// TIA Portal project "TesisIsitma_v1" (V19)

(* hardware
DEVICE "S7-1200 station_1"  S7-1200 Station
   slot 0: "Rack_0"  S7-1200 Rack  Rack  V1.0
   slot 1: "PLC_1"  CPU 1215C DC/DC/DC  6ES7 215-1AG40-0XB0  V4.5
*)

// ===== PLC "PLC_1"  CPU 1215C DC/DC/DC =====

VAR_GLOBAL   // PLC tag table "Default tag table"
   "System_Byte" AT %MB1 : Byte;
   "FirstScan" AT %M1.0 : Bool;
   "DiagStatusUpdate" AT %M1.1 : Bool;
   "AlwaysTRUE" AT %M1.2 : Bool;
   "AlwaysFALSE" AT %M1.3 : Bool;
   "Clock_Byte" AT %MB0 : Byte;
   "Clock_10Hz" AT %M0.0 : Bool;
   "Clock_5Hz" AT %M0.1 : Bool;
   "Clock_2.5Hz" AT %M0.2 : Bool;
   "Clock_2Hz" AT %M0.3 : Bool;
   "Clock_1.25Hz" AT %M0.4 : Bool;
   "Clock_1Hz" AT %M0.5 : Bool;
   "Clock_0.625Hz" AT %M0.6 : Bool;
   "Clock_0.5Hz" AT %M0.7 : Bool;
   "xSim" AT %M2.0 : Bool;
END_VAR

DATA_BLOCK "DB_Modbus"   // DB2
{ S7_Optimized_Access := 'FALSE' }
VERSION : 0.1
   VAR
      Req : Bool;
      Disconnect : Bool;
      Mode : USInt;
      DataAddress : UDInt := 40001;
      DataLength : UInt := 2;
      DataPointer : Array[0..3] of Byte;
      Connect : TCON_IP_v4;
   END_VAR
BEGIN
   Connect.RemoteAddress.ADDR[1] := 192;
   Connect.RemoteAddress.ADDR[2] := 168;
   Connect.RemoteAddress.ADDR[3] := 0;
   Connect.RemoteAddress.ADDR[4] := 48;
   Connect.InterfaceId := 64;
   Connect.ID := 6;
   Connect.RemotePort := 502;
   Connect.LocalPort := 502;
   Connect.ActiveEstablished := 1;
END_DATA_BLOCK

DATA_BLOCK "DB_Trig"   // DB3
{ S7_Optimized_Access := 'TRUE' }
VERSION : 0.1
   VAR
      "1" : Bool;
      "2" : Bool;
      "3" : Bool;
      "4" : Bool;
      "5" : Bool;
      "6" : Bool;
      "7" : Bool;
      "8" : Bool;
      "9" : Bool;
      "10" : Bool;
   END_VAR
BEGIN
END_DATA_BLOCK

ORGANIZATION_BLOCK "Main"   // OB1, LAD, ProgramCycle
TITLE = "Main Program Sweep (Cycle)"
{ S7_Optimized_Access := 'TRUE' }
VERSION : 0.1
   VAR_INPUT
      Initial_Call : Bool;   // Initial call of this OB
      Remanence : Bool;   // =True, if remanent data are available
   END_VAR
   VAR_TEMP   // added for the SCL form of the ladder/FBD networks
      _w1 : Bool;
      _w2 : Bool;
   END_VAR
BEGIN

REGION Network 1
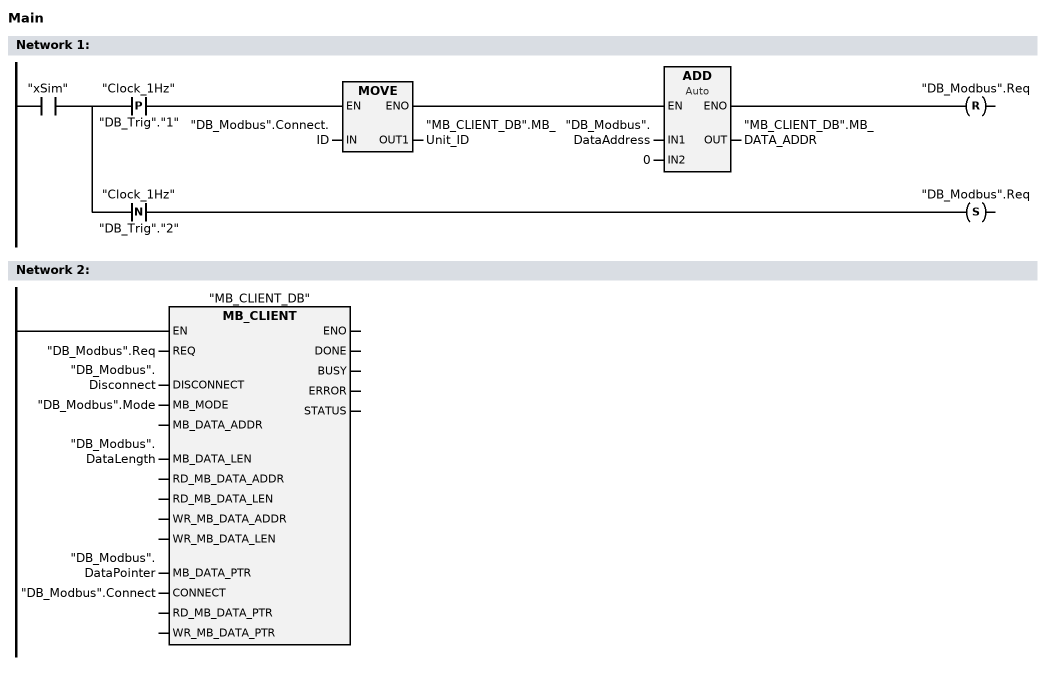
   RUNG wire#powerrail
      Contact( "xSim" )
      wire#w1
      P_Contact(operand := "Clock_1Hz", bit := "DB_Trig"."1")
      Move(in := "DB_Modbus".Connect.ID, out1 => "MB_CLIENT_DB".MB_Unit_ID)
      Add(in1 := "DB_Modbus".DataAddress, in2 := 0, out => "MB_CLIENT_DB".MB_DATA_ADDR)
      R_Coil( "DB_Modbus".Req )
   END_RUNG
   RUNG wire#w1
      N_Contact(operand := "Clock_1Hz", bit := "DB_Trig"."2")
      S_Coil( "DB_Modbus".Req )
   END_RUNG
   // the same network as SCL:
   #_w1 := "xSim" AND "Clock_1Hz" AND NOT "DB_Trig"."1";   // rising edge of "Clock_1Hz"
   "DB_Trig"."1" := "Clock_1Hz";
   IF #_w1 THEN
       "MB_CLIENT_DB".MB_Unit_ID := "DB_Modbus".Connect.ID;
       "MB_CLIENT_DB".MB_DATA_ADDR := "DB_Modbus".DataAddress + 0;
       "DB_Modbus".Req := FALSE;
   END_IF;
   #_w2 := "xSim" AND NOT "Clock_1Hz" AND "DB_Trig"."2";   // falling edge of "Clock_1Hz"
   "DB_Trig"."2" := "Clock_1Hz";
   IF #_w2 THEN "DB_Modbus".Req := TRUE; END_IF;
END_REGION

REGION Network 2
   "MB_CLIENT_DB"(REQ := "DB_Modbus".Req,   // MB_CLIENT
                  DISCONNECT := "DB_Modbus".Disconnect,
                  MB_MODE := "DB_Modbus".Mode,
                  MB_DATA_LEN := "DB_Modbus".DataLength,
                  MB_DATA_PTR := "DB_Modbus".DataPointer,
                  CONNECT := "DB_Modbus".Connect);
END_REGION
END_ORGANIZATION_BLOCK